PROGRAM FTP_CLIENT_DEMO
VAR
	FTP_CLIENT: FTP_CLIENT;
	ftp_activate: BOOL;
	ftp_done: BOOL;
	ftp_busy: BOOL;
	ftp_error_c: DWORD;
	ftp_error_t: BYTE;
	ftp_url: STRING := 'ftp://581920:123456@oscat.atwebpages.com:2000/subordner/';
	ftp_filename: STRING := '0100kb.bin';
	ftp_download: BOOL := TRUE;
	ftp_activ: BOOL := FALSE;
	file_delete: BOOL := FALSE;
	ftp_timeout: TIME := T#30s;
	zeit : TIME := T#30s;
	stop: BOOL;
	start: BOOL :=TRUE ;
	reset: BOOL;
	error: DWORD;
	ok: DWORD;
	CLK_PRG_1: CLK_PRG;
	COUNT_DR_1: COUNT_DR;
	COUNT_DR_2: COUNT_DR;
END_VAR
VAR // added by the converter: edge detectors and wires of the graphical bodies
    _w1, _w2 : ANY;
END_VAR

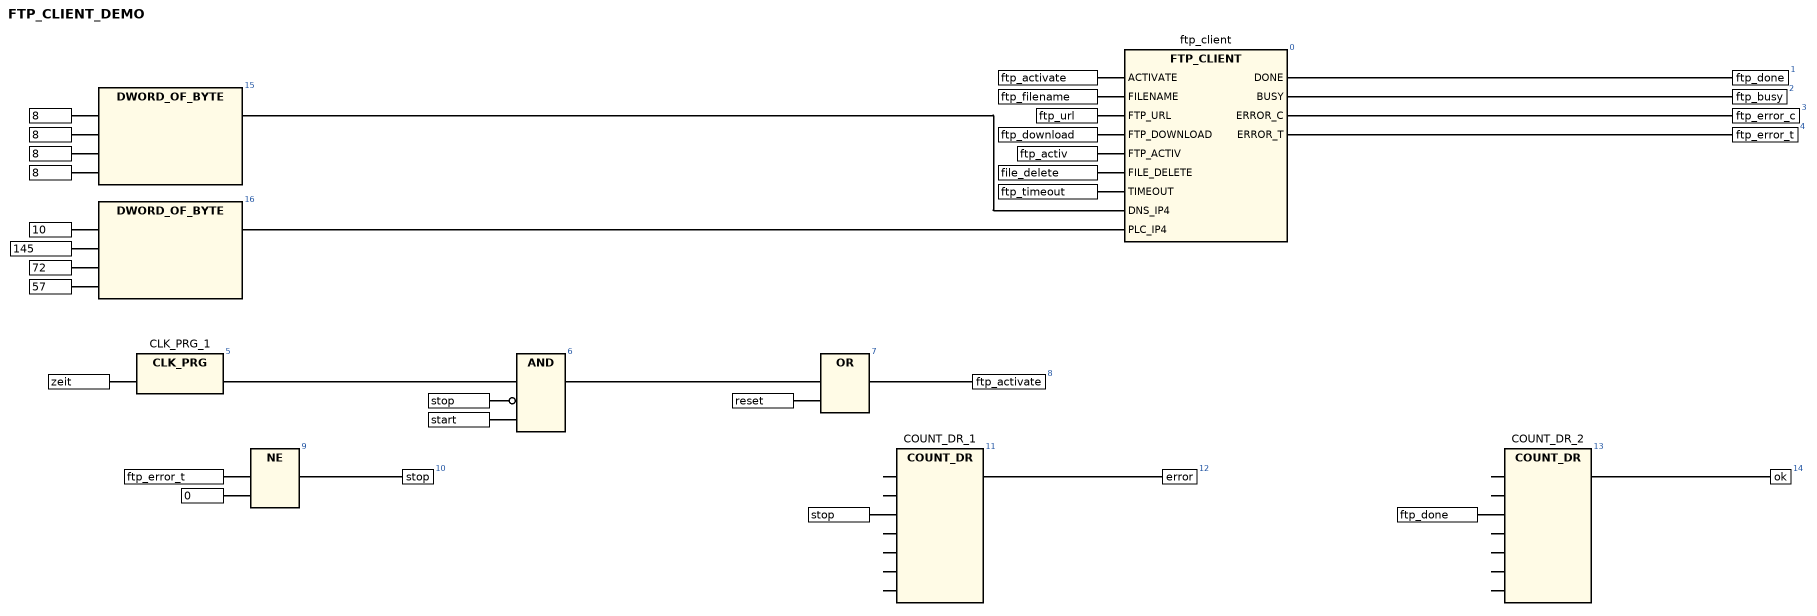
ftp_client(
    ACTIVATE := ftp_activate,
    FILENAME := ftp_filename,
    FTP_URL := ftp_url,
    FTP_DOWNLOAD := ftp_download,
    FTP_ACTIV := ftp_activ,
    FILE_DELETE := file_delete,
    TIMEOUT := ftp_timeout,
    DNS_IP4 := _w1,
    PLC_IP4 := _w2);
ftp_done := ftp_client.DONE;
ftp_busy := ftp_client.BUSY;
ftp_error_c := ftp_client.ERROR_C;
ftp_error_t := ftp_client.ERROR_T;
CLK_PRG_1(_in1 := zeit); // CLK_PRG
ftp_activate := CLK_PRG_1._out1 AND NOT stop AND start OR reset;
stop := ftp_error_t <> 0;
COUNT_DR_1(_in3 := stop); // COUNT_DR
error := COUNT_DR_1._out1;
COUNT_DR_2(_in3 := ftp_done); // COUNT_DR
ok := COUNT_DR_2._out1;
_w1 := DWORD_OF_BYTE(8, 8, 8, 8);
_w2 := DWORD_OF_BYTE(10, 145, 72, 57);

END_PROGRAM

(* stored: Version 1.1.0.1, ProductVersion 3.1.4022.7
   POU FTP_CLIENT_DEMO: Id {2f67d7d6-7b93-4e1d-9029-c142b1f7d9c3}, SpecialFunc None *)
